INTERFACE I_XtsTrack

PROPERTY TrackLength : MC_Lreal
GET
END_GET
END_PROPERTY

END_INTERFACE

(* stored: Version 1.1.0.1, ProductVersion 3.1.4024.12
   Itf I_XtsTrack: Id {b580e084-f2aa-4b9e-b34b-5773df679de5}
   Property TrackLength: Id {d09b154e-641d-4452-b45a-353375f2a798}
   Get Get: Id {227be027-fd95-4a28-b451-be32068fa3af} *)
